// TIA Portal V16 export
// export: Created 2021-11-12T13:31:54.5417343Z, ExportSetting WithDefaults, DisplayName Totally Integrated Automation Portal, DisplayVersion V16 Update 3, DisplayName TIA Portal Version Control Interface, DisplayVersion V16 Update 2, DisplayName TIA Portal Openness, DisplayVersion V16 Update 3, DisplayName SINAMICS Startdrive Advanced, DisplayVersion V16 Update 5, DisplayName SINAMICS Startdrive G130, G150, S120, S150, SINAMICS MV, S210, DisplayVersion V16 Update 5, DisplayName SINAMICS Startdrive G110M, G120, G120C, G120D, G120P, G115D, DisplayVersion V16 Update 5, DisplayName STEP 7 Professional, DisplayVersion V16 Update 3, DisplayName STEP 7 Safety, DisplayVersion V16, DisplayName WinCC UA Professional, DisplayVersion V16 Update 3
FUNCTION_BLOCK "Cab_000+UC10"   // FB75, LAD
TITLE = FB Cabinet V1.01
{ S7_Optimized_Access := 'TRUE' }
VERSION : 0.1
// MICE Wood block
// Cabinet V1.01
// functionality regarding cabinet, like errors from main switch, circuit breakers, temperature in cabinet,……
// stored: AutoNumber true, IsIECCheckEnabled false, IsRetainMemResEnabled false, MemoryReserve 100, SetENOAutomatically false, UDAEnableTagReadback false
   VAR
      "SF_UC10-FV01_11_Alarm" { S7_SetPoint := 'True'} : "STD_DI_Mon";
      "SF_UC10-FB21_14_Alarm" { S7_SetPoint := 'True'} : "STD_DI_Mon";
      "SF_UC10-FC21_14_Alarm" { S7_SetPoint := 'True'} : "STD_DI_Mon";
      "SF_UC10-EC01_3_Alarm" { S7_SetPoint := 'True'} : "STD_DI_Mon";
      "SF_UC10-FC01_14_Alarm" { S7_SetPoint := 'True'} : "STD_DI_Mon";
      "SF_UC10-TB01_14_Alarm" { S7_SetPoint := 'True'} : "STD_DI_Mon";
      "SF_UC10-FC30_14_Alarm" { S7_SetPoint := 'True'} : "STD_DI_Mon";
      "SF_UC10-FC30_24_Alarm" { S7_SetPoint := 'True'} : "STD_DI_Mon";
      "SF_UC10-FC50_14_Alarm" { S7_SetPoint := 'True'} : "STD_DI_Mon";
      "SF_UC10-FC51_24_Alarm" { S7_SetPoint := 'True'} : "STD_DI_Mon";
      "SF_UC12-FC21_14_Alarm" { S7_SetPoint := 'True'} : "STD_DI_Mon";
      "SF_UC12-EC01_3_Alarm" { S7_SetPoint := 'True'} : "STD_DI_Mon";
      "SF_UC11-FC01_14_Alarm" { S7_SetPoint := 'True'} : "STD_DI_Mon";
      "SF_UC11-FC02_14_Alarm" { S7_SetPoint := 'True'} : "STD_DI_Mon";
      "SF_UC11-FC03_14_Alarm" { S7_SetPoint := 'True'} : "STD_DI_Mon";
   END_VAR
   VAR_TEMP
      TB1Ack : Bool;
      TB1Aux : Bool;
   END_VAR
   VAR_TEMP   // added for the SCL form of the ladder/FBD networks
      _w1 : Bool;
      _w2 : Bool;
      _w3 : Bool;
      _w4 : Bool;
      _w5 : Bool;
      _w6 : Bool;
      _w7 : Bool;
   END_VAR
BEGIN

REGION Network 1: Aknowledge logic - Any zone can acknowledge alarms
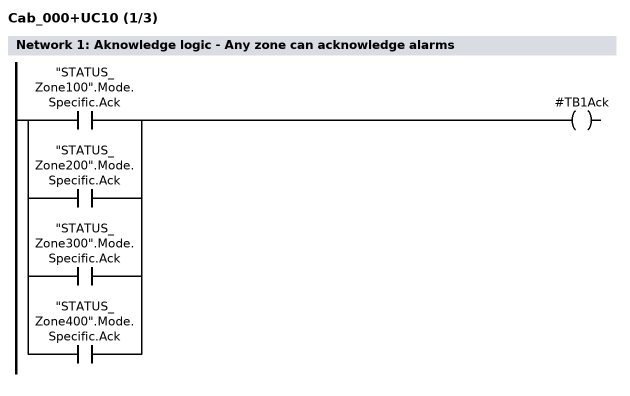
   RUNG wire#powerrail
      Contact( "STATUS_Zone100".Mode.Specific.Ack )
      wire#w1
      Coil( #TB1Ack )
   END_RUNG
   RUNG wire#powerrail
      Contact( "STATUS_Zone200".Mode.Specific.Ack )
   END_RUNG wire#w1
   RUNG wire#powerrail
      Contact( "STATUS_Zone300".Mode.Specific.Ack )
   END_RUNG wire#w1
   RUNG wire#powerrail
      Contact( "STATUS_Zone400".Mode.Specific.Ack )
   END_RUNG wire#w1
   // the same network as SCL:
   #TB1Ack := "STATUS_Zone100".Mode.Specific.Ack OR "STATUS_Zone200".Mode.Specific.Ack OR "STATUS_Zone300".Mode.Specific.Ack OR "STATUS_Zone400".Mode.Specific.Ack;
END_REGION

REGION Network 2: ************************* Alarms ******************************
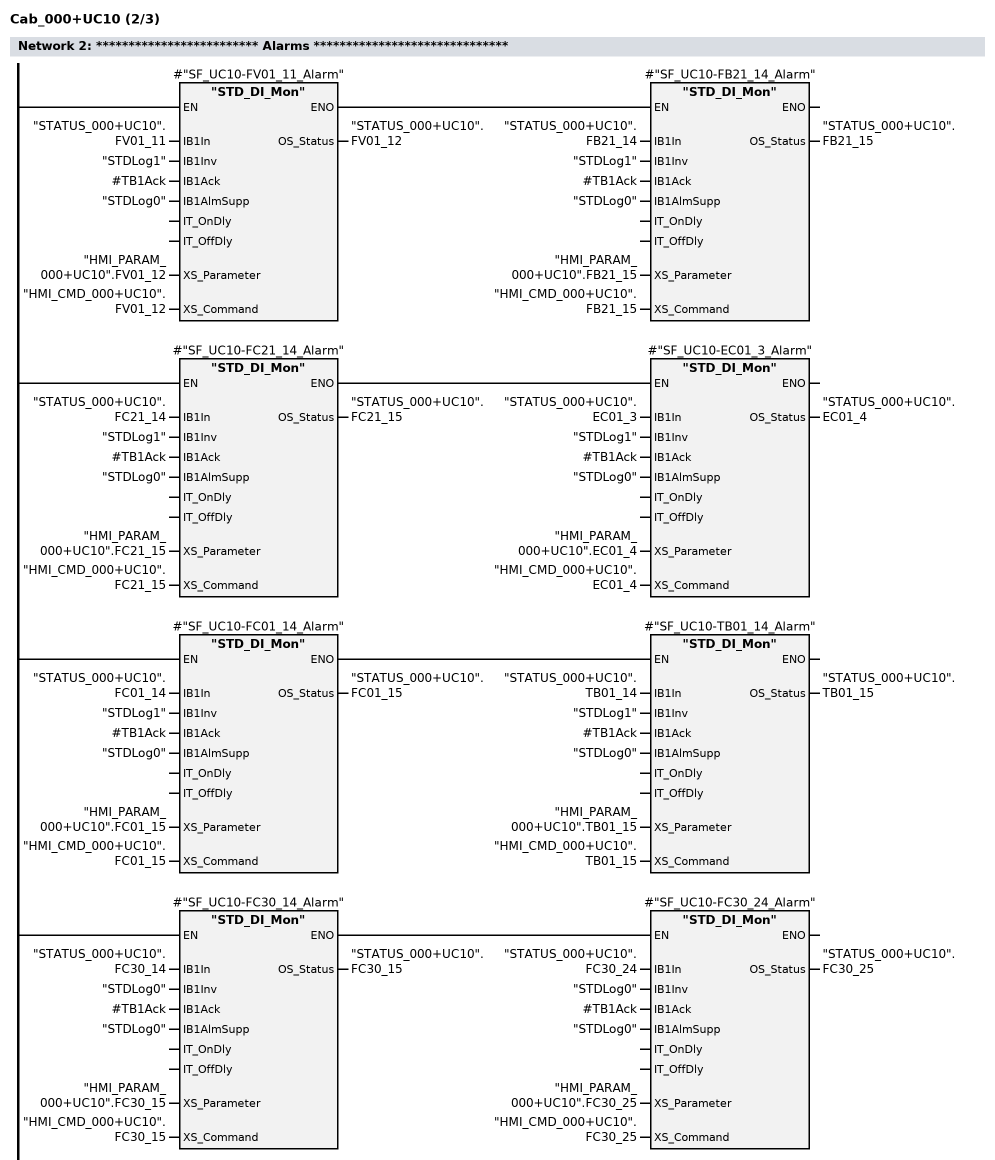
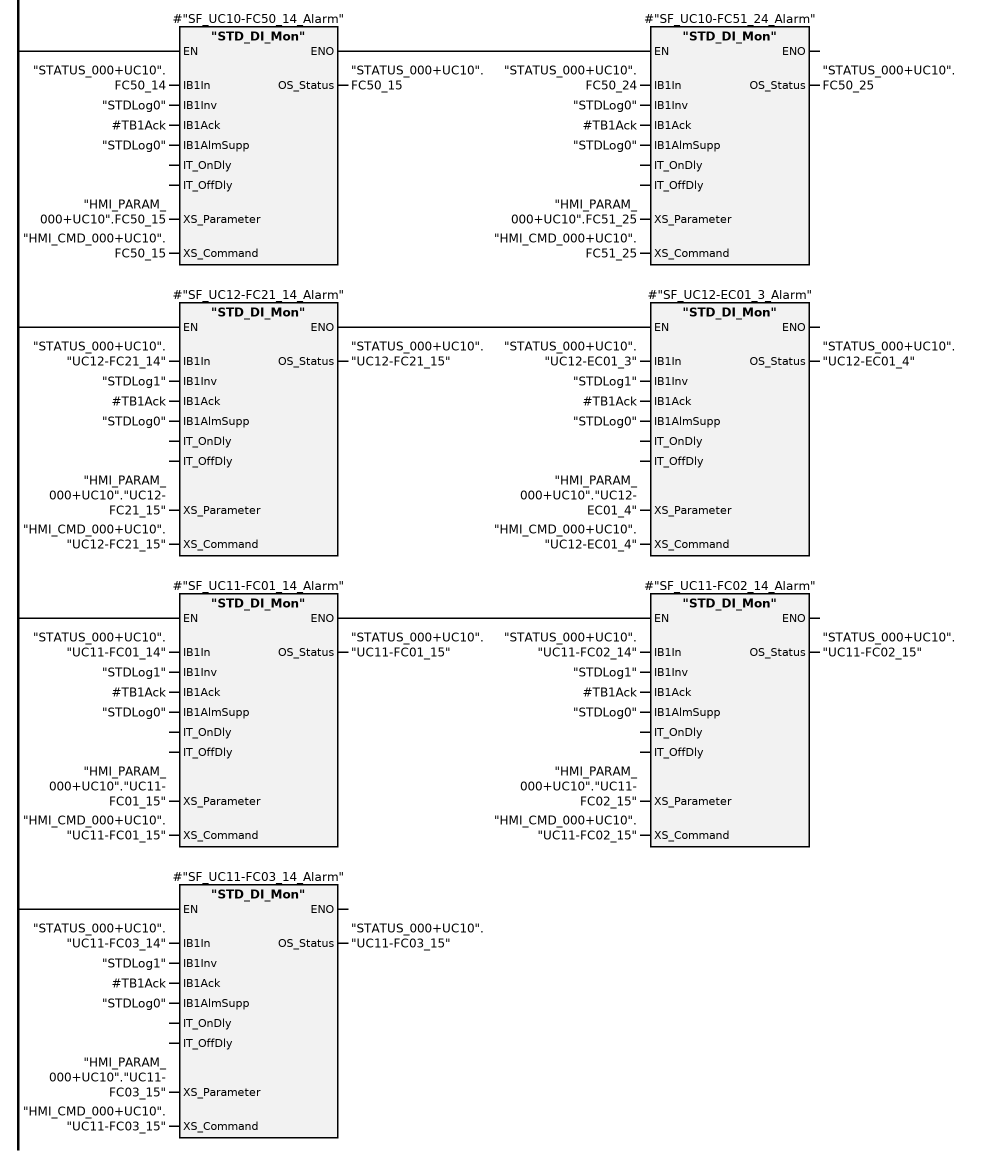
   RUNG wire#powerrail
      #"SF_UC10-FV01_11_Alarm"(IB1In := "STATUS_000+UC10".FV01_11, IB1Inv := "STDLog1", IB1Ack := #TB1Ack, IB1AlmSupp := "STDLog0", IT_OnDly :=, IT_OffDly :=, XS_Parameter := "HMI_PARAM_000+UC10".FV01_12, XS_Command := "HMI_CMD_000+UC10".FV01_12, OS_Status => "STATUS_000+UC10".FV01_12)
      #"SF_UC10-FB21_14_Alarm"(IB1In := "STATUS_000+UC10".FB21_14, IB1Inv := "STDLog1", IB1Ack := #TB1Ack, IB1AlmSupp := "STDLog0", IT_OnDly :=, IT_OffDly :=, XS_Parameter := "HMI_PARAM_000+UC10".FB21_15, XS_Command := "HMI_CMD_000+UC10".FB21_15, OS_Status => "STATUS_000+UC10".FB21_15)
   END_RUNG
   RUNG wire#powerrail
      #"SF_UC10-FC21_14_Alarm"(IB1In := "STATUS_000+UC10".FC21_14, IB1Inv := "STDLog1", IB1Ack := #TB1Ack, IB1AlmSupp := "STDLog0", IT_OnDly :=, IT_OffDly :=, XS_Parameter := "HMI_PARAM_000+UC10".FC21_15, XS_Command := "HMI_CMD_000+UC10".FC21_15, OS_Status => "STATUS_000+UC10".FC21_15)
      #"SF_UC10-EC01_3_Alarm"(IB1In := "STATUS_000+UC10".EC01_3, IB1Inv := "STDLog1", IB1Ack := #TB1Ack, IB1AlmSupp := "STDLog0", IT_OnDly :=, IT_OffDly :=, XS_Parameter := "HMI_PARAM_000+UC10".EC01_4, XS_Command := "HMI_CMD_000+UC10".EC01_4, OS_Status => "STATUS_000+UC10".EC01_4)
   END_RUNG
   RUNG wire#powerrail
      #"SF_UC10-FC01_14_Alarm"(IB1In := "STATUS_000+UC10".FC01_14, IB1Inv := "STDLog1", IB1Ack := #TB1Ack, IB1AlmSupp := "STDLog0", IT_OnDly :=, IT_OffDly :=, XS_Parameter := "HMI_PARAM_000+UC10".FC01_15, XS_Command := "HMI_CMD_000+UC10".FC01_15, OS_Status => "STATUS_000+UC10".FC01_15)
      #"SF_UC10-TB01_14_Alarm"(IB1In := "STATUS_000+UC10".TB01_14, IB1Inv := "STDLog1", IB1Ack := #TB1Ack, IB1AlmSupp := "STDLog0", IT_OnDly :=, IT_OffDly :=, XS_Parameter := "HMI_PARAM_000+UC10".TB01_15, XS_Command := "HMI_CMD_000+UC10".TB01_15, OS_Status => "STATUS_000+UC10".TB01_15)
   END_RUNG
   RUNG wire#powerrail
      #"SF_UC10-FC30_14_Alarm"(IB1In := "STATUS_000+UC10".FC30_14, IB1Inv := "STDLog0", IB1Ack := #TB1Ack, IB1AlmSupp := "STDLog0", IT_OnDly :=, IT_OffDly :=, XS_Parameter := "HMI_PARAM_000+UC10".FC30_15, XS_Command := "HMI_CMD_000+UC10".FC30_15, OS_Status => "STATUS_000+UC10".FC30_15)
      #"SF_UC10-FC30_24_Alarm"(IB1In := "STATUS_000+UC10".FC30_24, IB1Inv := "STDLog0", IB1Ack := #TB1Ack, IB1AlmSupp := "STDLog0", IT_OnDly :=, IT_OffDly :=, XS_Parameter := "HMI_PARAM_000+UC10".FC30_25, XS_Command := "HMI_CMD_000+UC10".FC30_25, OS_Status => "STATUS_000+UC10".FC30_25)
   END_RUNG
   RUNG wire#powerrail
      #"SF_UC10-FC50_14_Alarm"(IB1In := "STATUS_000+UC10".FC50_14, IB1Inv := "STDLog0", IB1Ack := #TB1Ack, IB1AlmSupp := "STDLog0", IT_OnDly :=, IT_OffDly :=, XS_Parameter := "HMI_PARAM_000+UC10".FC50_15, XS_Command := "HMI_CMD_000+UC10".FC50_15, OS_Status => "STATUS_000+UC10".FC50_15)
      #"SF_UC10-FC51_24_Alarm"(IB1In := "STATUS_000+UC10".FC50_24, IB1Inv := "STDLog0", IB1Ack := #TB1Ack, IB1AlmSupp := "STDLog0", IT_OnDly :=, IT_OffDly :=, XS_Parameter := "HMI_PARAM_000+UC10".FC51_25, XS_Command := "HMI_CMD_000+UC10".FC51_25, OS_Status => "STATUS_000+UC10".FC50_25)
   END_RUNG
   RUNG wire#powerrail
      #"SF_UC12-FC21_14_Alarm"(IB1In := "STATUS_000+UC10"."UC12-FC21_14", IB1Inv := "STDLog1", IB1Ack := #TB1Ack, IB1AlmSupp := "STDLog0", IT_OnDly :=, IT_OffDly :=, XS_Parameter := "HMI_PARAM_000+UC10"."UC12-FC21_15", XS_Command := "HMI_CMD_000+UC10"."UC12-FC21_15", OS_Status => "STATUS_000+UC10"."UC12-FC21_15")
      #"SF_UC12-EC01_3_Alarm"(IB1In := "STATUS_000+UC10"."UC12-EC01_3", IB1Inv := "STDLog1", IB1Ack := #TB1Ack, IB1AlmSupp := "STDLog0", IT_OnDly :=, IT_OffDly :=, XS_Parameter := "HMI_PARAM_000+UC10"."UC12-EC01_4", XS_Command := "HMI_CMD_000+UC10"."UC12-EC01_4", OS_Status => "STATUS_000+UC10"."UC12-EC01_4")
   END_RUNG
   RUNG wire#powerrail
      #"SF_UC11-FC01_14_Alarm"(IB1In := "STATUS_000+UC10"."UC11-FC01_14", IB1Inv := "STDLog1", IB1Ack := #TB1Ack, IB1AlmSupp := "STDLog0", IT_OnDly :=, IT_OffDly :=, XS_Parameter := "HMI_PARAM_000+UC10"."UC11-FC01_15", XS_Command := "HMI_CMD_000+UC10"."UC11-FC01_15", OS_Status => "STATUS_000+UC10"."UC11-FC01_15")
      #"SF_UC11-FC02_14_Alarm"(IB1In := "STATUS_000+UC10"."UC11-FC02_14", IB1Inv := "STDLog1", IB1Ack := #TB1Ack, IB1AlmSupp := "STDLog0", IT_OnDly :=, IT_OffDly :=, XS_Parameter := "HMI_PARAM_000+UC10"."UC11-FC02_15", XS_Command := "HMI_CMD_000+UC10"."UC11-FC02_15", OS_Status => "STATUS_000+UC10"."UC11-FC02_15")
   END_RUNG
   RUNG wire#powerrail
      #"SF_UC11-FC03_14_Alarm"(IB1In := "STATUS_000+UC10"."UC11-FC03_14", IB1Inv := "STDLog1", IB1Ack := #TB1Ack, IB1AlmSupp := "STDLog0", IT_OnDly :=, IT_OffDly :=, XS_Parameter := "HMI_PARAM_000+UC10"."UC11-FC03_15", XS_Command := "HMI_CMD_000+UC10"."UC11-FC03_15", OS_Status => "STATUS_000+UC10"."UC11-FC03_15")
   END_RUNG
   // the same network as SCL:
   #"SF_UC10-FV01_11_Alarm"(IB1In := "STATUS_000+UC10".FV01_11,   // "STD_DI_Mon"
                           IB1Inv := "STDLog1",
                           IB1Ack := #TB1Ack,
                           IB1AlmSupp := "STDLog0",
                           XS_Parameter := "HMI_PARAM_000+UC10".FV01_12,
                           XS_Command := "HMI_CMD_000+UC10".FV01_12,
                           OS_Status => "STATUS_000+UC10".FV01_12,
                           ENO => #_w1);
   IF #_w1 THEN
       #"SF_UC10-FB21_14_Alarm"(IB1In := "STATUS_000+UC10".FB21_14,   // "STD_DI_Mon"
                               IB1Inv := "STDLog1",
                               IB1Ack := #TB1Ack,
                               IB1AlmSupp := "STDLog0",
                               XS_Parameter := "HMI_PARAM_000+UC10".FB21_15,
                               XS_Command := "HMI_CMD_000+UC10".FB21_15,
                               OS_Status => "STATUS_000+UC10".FB21_15);
   END_IF;
   #"SF_UC10-FC21_14_Alarm"(IB1In := "STATUS_000+UC10".FC21_14,   // "STD_DI_Mon"
                           IB1Inv := "STDLog1",
                           IB1Ack := #TB1Ack,
                           IB1AlmSupp := "STDLog0",
                           XS_Parameter := "HMI_PARAM_000+UC10".FC21_15,
                           XS_Command := "HMI_CMD_000+UC10".FC21_15,
                           OS_Status => "STATUS_000+UC10".FC21_15,
                           ENO => #_w2);
   IF #_w2 THEN
       #"SF_UC10-EC01_3_Alarm"(IB1In := "STATUS_000+UC10".EC01_3,   // "STD_DI_Mon"
                               IB1Inv := "STDLog1",
                               IB1Ack := #TB1Ack,
                               IB1AlmSupp := "STDLog0",
                               XS_Parameter := "HMI_PARAM_000+UC10".EC01_4,
                               XS_Command := "HMI_CMD_000+UC10".EC01_4,
                               OS_Status => "STATUS_000+UC10".EC01_4);
   END_IF;
   #"SF_UC10-FC01_14_Alarm"(IB1In := "STATUS_000+UC10".FC01_14,   // "STD_DI_Mon"
                           IB1Inv := "STDLog1",
                           IB1Ack := #TB1Ack,
                           IB1AlmSupp := "STDLog0",
                           XS_Parameter := "HMI_PARAM_000+UC10".FC01_15,
                           XS_Command := "HMI_CMD_000+UC10".FC01_15,
                           OS_Status => "STATUS_000+UC10".FC01_15,
                           ENO => #_w3);
   IF #_w3 THEN
       #"SF_UC10-TB01_14_Alarm"(IB1In := "STATUS_000+UC10".TB01_14,   // "STD_DI_Mon"
                               IB1Inv := "STDLog1",
                               IB1Ack := #TB1Ack,
                               IB1AlmSupp := "STDLog0",
                               XS_Parameter := "HMI_PARAM_000+UC10".TB01_15,
                               XS_Command := "HMI_CMD_000+UC10".TB01_15,
                               OS_Status => "STATUS_000+UC10".TB01_15);
   END_IF;
   #"SF_UC10-FC30_14_Alarm"(IB1In := "STATUS_000+UC10".FC30_14,   // "STD_DI_Mon"
                           IB1Inv := "STDLog0",
                           IB1Ack := #TB1Ack,
                           IB1AlmSupp := "STDLog0",
                           XS_Parameter := "HMI_PARAM_000+UC10".FC30_15,
                           XS_Command := "HMI_CMD_000+UC10".FC30_15,
                           OS_Status => "STATUS_000+UC10".FC30_15,
                           ENO => #_w4);
   IF #_w4 THEN
       #"SF_UC10-FC30_24_Alarm"(IB1In := "STATUS_000+UC10".FC30_24,   // "STD_DI_Mon"
                               IB1Inv := "STDLog0",
                               IB1Ack := #TB1Ack,
                               IB1AlmSupp := "STDLog0",
                               XS_Parameter := "HMI_PARAM_000+UC10".FC30_25,
                               XS_Command := "HMI_CMD_000+UC10".FC30_25,
                               OS_Status => "STATUS_000+UC10".FC30_25);
   END_IF;
   #"SF_UC10-FC50_14_Alarm"(IB1In := "STATUS_000+UC10".FC50_14,   // "STD_DI_Mon"
                           IB1Inv := "STDLog0",
                           IB1Ack := #TB1Ack,
                           IB1AlmSupp := "STDLog0",
                           XS_Parameter := "HMI_PARAM_000+UC10".FC50_15,
                           XS_Command := "HMI_CMD_000+UC10".FC50_15,
                           OS_Status => "STATUS_000+UC10".FC50_15,
                           ENO => #_w5);
   IF #_w5 THEN
       #"SF_UC10-FC51_24_Alarm"(IB1In := "STATUS_000+UC10".FC50_24,   // "STD_DI_Mon"
                               IB1Inv := "STDLog0",
                               IB1Ack := #TB1Ack,
                               IB1AlmSupp := "STDLog0",
                               XS_Parameter := "HMI_PARAM_000+UC10".FC51_25,
                               XS_Command := "HMI_CMD_000+UC10".FC51_25,
                               OS_Status => "STATUS_000+UC10".FC50_25);
   END_IF;
   #"SF_UC12-FC21_14_Alarm"(IB1In := "STATUS_000+UC10"."UC12-FC21_14",   // "STD_DI_Mon"
                           IB1Inv := "STDLog1",
                           IB1Ack := #TB1Ack,
                           IB1AlmSupp := "STDLog0",
                           XS_Parameter := "HMI_PARAM_000+UC10"."UC12-FC21_15",
                           XS_Command := "HMI_CMD_000+UC10"."UC12-FC21_15",
                           OS_Status => "STATUS_000+UC10"."UC12-FC21_15",
                           ENO => #_w6);
   IF #_w6 THEN
       #"SF_UC12-EC01_3_Alarm"(IB1In := "STATUS_000+UC10"."UC12-EC01_3",   // "STD_DI_Mon"
                               IB1Inv := "STDLog1",
                               IB1Ack := #TB1Ack,
                               IB1AlmSupp := "STDLog0",
                               XS_Parameter := "HMI_PARAM_000+UC10"."UC12-EC01_4",
                               XS_Command := "HMI_CMD_000+UC10"."UC12-EC01_4",
                               OS_Status => "STATUS_000+UC10"."UC12-EC01_4");
   END_IF;
   #"SF_UC11-FC01_14_Alarm"(IB1In := "STATUS_000+UC10"."UC11-FC01_14",   // "STD_DI_Mon"
                           IB1Inv := "STDLog1",
                           IB1Ack := #TB1Ack,
                           IB1AlmSupp := "STDLog0",
                           XS_Parameter := "HMI_PARAM_000+UC10"."UC11-FC01_15",
                           XS_Command := "HMI_CMD_000+UC10"."UC11-FC01_15",
                           OS_Status => "STATUS_000+UC10"."UC11-FC01_15",
                           ENO => #_w7);
   IF #_w7 THEN
       #"SF_UC11-FC02_14_Alarm"(IB1In := "STATUS_000+UC10"."UC11-FC02_14",   // "STD_DI_Mon"
                               IB1Inv := "STDLog1",
                               IB1Ack := #TB1Ack,
                               IB1AlmSupp := "STDLog0",
                               XS_Parameter := "HMI_PARAM_000+UC10"."UC11-FC02_15",
                               XS_Command := "HMI_CMD_000+UC10"."UC11-FC02_15",
                               OS_Status => "STATUS_000+UC10"."UC11-FC02_15");
   END_IF;
   #"SF_UC11-FC03_14_Alarm"(IB1In := "STATUS_000+UC10"."UC11-FC03_14",   // "STD_DI_Mon"
                           IB1Inv := "STDLog1",
                           IB1Ack := #TB1Ack,
                           IB1AlmSupp := "STDLog0",
                           XS_Parameter := "HMI_PARAM_000+UC10"."UC11-FC03_15",
                           XS_Command := "HMI_CMD_000+UC10"."UC11-FC03_15",
                           OS_Status => "STATUS_000+UC10"."UC11-FC03_15");
END_REGION

REGION Network 3: Sum of significant alarms
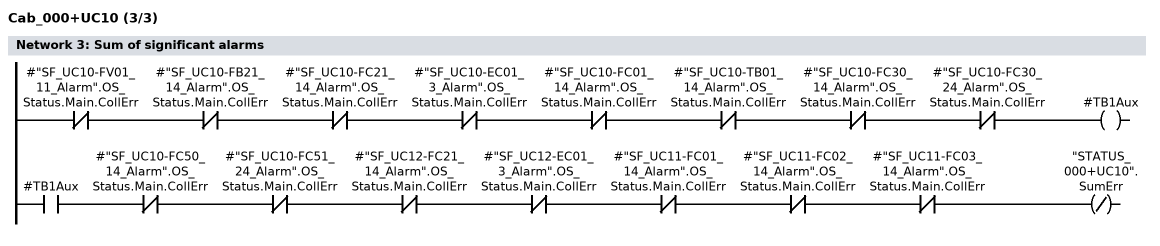
   RUNG wire#powerrail
      I_Contact( #"SF_UC10-FV01_11_Alarm".OS_Status.Main.CollErr )
      I_Contact( #"SF_UC10-FB21_14_Alarm".OS_Status.Main.CollErr )
      I_Contact( #"SF_UC10-FC21_14_Alarm".OS_Status.Main.CollErr )
      I_Contact( #"SF_UC10-EC01_3_Alarm".OS_Status.Main.CollErr )
      I_Contact( #"SF_UC10-FC01_14_Alarm".OS_Status.Main.CollErr )
      I_Contact( #"SF_UC10-TB01_14_Alarm".OS_Status.Main.CollErr )
      I_Contact( #"SF_UC10-FC30_14_Alarm".OS_Status.Main.CollErr )
      I_Contact( #"SF_UC10-FC30_24_Alarm".OS_Status.Main.CollErr )
      Coil( #TB1Aux )
   END_RUNG
   RUNG wire#powerrail
      Contact( #TB1Aux )
      I_Contact( #"SF_UC10-FC50_14_Alarm".OS_Status.Main.CollErr )
      I_Contact( #"SF_UC10-FC51_24_Alarm".OS_Status.Main.CollErr )
      I_Contact( #"SF_UC12-FC21_14_Alarm".OS_Status.Main.CollErr )
      I_Contact( #"SF_UC12-EC01_3_Alarm".OS_Status.Main.CollErr )
      I_Contact( #"SF_UC11-FC01_14_Alarm".OS_Status.Main.CollErr )
      I_Contact( #"SF_UC11-FC02_14_Alarm".OS_Status.Main.CollErr )
      I_Contact( #"SF_UC11-FC03_14_Alarm".OS_Status.Main.CollErr )
      I_Coil( "STATUS_000+UC10".SumErr )
   END_RUNG
   // the same network as SCL:
   #TB1Aux := NOT #"SF_UC10-FV01_11_Alarm".OS_Status.Main.CollErr AND NOT #"SF_UC10-FB21_14_Alarm".OS_Status.Main.CollErr AND NOT #"SF_UC10-FC21_14_Alarm".OS_Status.Main.CollErr AND NOT #"SF_UC10-EC01_3_Alarm".OS_Status.Main.CollErr AND NOT #"SF_UC10-FC01_14_Alarm".OS_Status.Main.CollErr AND NOT #"SF_UC10-TB01_14_Alarm".OS_Status.Main.CollErr AND NOT #"SF_UC10-FC30_14_Alarm".OS_Status.Main.CollErr AND NOT #"SF_UC10-FC30_24_Alarm".OS_Status.Main.CollErr;
   "STATUS_000+UC10".SumErr := NOT (#TB1Aux AND NOT #"SF_UC10-FC50_14_Alarm".OS_Status.Main.CollErr AND NOT #"SF_UC10-FC51_24_Alarm".OS_Status.Main.CollErr AND NOT #"SF_UC12-FC21_14_Alarm".OS_Status.Main.CollErr AND NOT #"SF_UC12-EC01_3_Alarm".OS_Status.Main.CollErr AND NOT #"SF_UC11-FC01_14_Alarm".OS_Status.Main.CollErr AND NOT #"SF_UC11-FC02_14_Alarm".OS_Status.Main.CollErr AND NOT #"SF_UC11-FC03_14_Alarm".OS_Status.Main.CollErr);
END_REGION

REGION Network 4: Significant voltage OK
END_REGION
END_FUNCTION_BLOCK
